// TIA Portal V17 export
// export: Created 2022-07-20T07:01:33.194346Z, ExportSetting WithDefaults, DisplayName Totally Integrated Automation Portal, DisplayVersion V17, DisplayName TIA Portal Openness, DisplayVersion V17, DisplayName TIA Portal Version Control Interface, DisplayVersion V17, DisplayName SINAMICS Startdrive Advanced, DisplayVersion V17, DisplayName SINAMICS Startdrive G130, G150, S120, S150, SINAMICS MV, S210, DisplayVersion V17, DisplayName SINAMICS Startdrive G110M, G120, G120C, G120D, G120P, G115D, DisplayVersion V17, DisplayName STEP 7 Professional, DisplayVersion V17, DisplayName STEP 7 Safety, DisplayVersion V17, DisplayName WinCC Advanced, DisplayVersion V17
FUNCTION_BLOCK "FB10321_CompactPrintingHeadsTray"   // FB10321, LAD
{ S7_Optimized_Access := 'TRUE' }
VERSION : 0.1
// stored: AutoNumber false, IsIECCheckEnabled false, IsRetainMemResEnabled false, MemoryReserve 100, SetENOAutomatically false, UDAEnableTagReadback false
   VAR_INPUT
      HeadsTray_RequestHeadsTraySafetyPosition : Bool;
      VerticalMotor_OriginPosition : Real;
      VerticalMotor_CleaningPosition : Real;
      VerticalMotor_WipingPosition : Real;
      VerticalMotor_PurgePosition : Real;
      VerticalMotor_PrintingPosition : Real;
      "VerticalMotor_Velocity_mm.s-1" : Real;
      VerticalMotor_ScaleInverted : Bool;
      HorizontalMotor_OriginPosition : Real;
      HorizontalMotor_WipingPosition : Real;
      HorizontalMotor_PurgePosition : Real;
      HorizontalMotor_Heads12Position : Real;
      HorizontalMotor_Heads34Position : Real;
      HorizontalMotor_Heads56Position : Real;
      HorizontalMotor_PrintingPosition : Real;
      "HorizontalMotor_Velocity_mm.s-1" : Real;
      HorizontalMotor_ScaleInverted : Bool;
      VerticalMotorDrive_In : "TLexium_MDrv_Drv2Plc";
      HorizontalMotorDrive_In : "TLexium_MDrv_Drv2Plc";
   END_VAR
   VAR_OUTPUT
      VerticalMotor_ActualPosition_mm : Real;
      HorizontalMotor_ActualPosition_mm : Real;
      HeadsTray_HomingDone : Bool;
      HeadsTray_IsInSafetyPosition : Bool;
      HeadsTray_IsInOriginPosition : Bool;
      HeadsTray_IsInHeads12CleaningPosition : Bool;
      HeadsTray_IsInHeads34CleaningPosition : Bool;
      HeadsTray_IsInHeads56CleaningPosition : Bool;
      HeadsTray_IsInWipingPosition : Bool;
      HeadsTray_IsInPurgePosition : Bool;
      HeadsTray_IsInHighPosition : Bool;
      HeadsTray_IsInPrintingPosition : Bool;
      HorizontalMotor_IsInOriginPosition : Bool;
      HorizontalMotor_IsInPurgePosition : Bool;
      HorizontalMotor_IsInWipingPosition : Bool;
      HorizontalMotor_IsInHeads12Position : Bool;
      HorizontalMotor_IsInHeads34Position : Bool;
      HorizontalMotor_IsInHeads56Position : Bool;
      HorizontalMotor_IsInPrintingPosition : Bool;
      VerticalMotor_IsInOriginPosition : Bool;
      VerticalMotor_IsInCleaningPosition : Bool;
      VerticalMotor_IsInWipingPosition : Bool;
      VerticalMotor_IsInPurgePosition : Bool;
      VerticalMotor_IsInPrintingPosition : Bool;
      SuccionDisk : Bool;
      VerticalMotor_InError : Bool;
      VerticalMotor_ErrorCode : Array[0..9] of UInt;
      HorizontalMotor_InError : Bool;
      HorizontalMotor_ErrorCode : Array[0..9] of UInt;
   END_VAR
   VAR_IN_OUT
      VerticalMotorDrive_Out : "TLexium_MDrv_Plc2Drv";
      HorizontalMotorDrive_Out : "TLexium_MDrv_Plc2Drv";
      RequestAcknowledge : Bool;
      RequestHoming : Bool;
      RequestStop : Bool;
      RequestGoToOriginPosition : Bool;
      RequestGoToWipingPosition : Bool;
      RequestGoToPurgePosition : Bool;
      RequestGoToHorizontalHeads12Position : Bool;
      RequestGoToHorizontalHeads34Position : Bool;
      RequestGoToHorizontalHeads56Position : Bool;
      RequestGoToVerticalOriginPosition : Bool;
      RequestGoToVerticalCleaningPosition : Bool;
      RequestGoToHighPosition : Bool;
      RequestGoToPrintingPosition : Bool;
   END_VAR
   VAR
      HeadsTrayMovementStateDiagram : Int;
      HeadsTraySafetyMovementStateDiagram : Int;
      R_TRIG_RequestHoming : R_TRIG;
      R_TRIG_RequestGoToOriginPosition { S7_SetPoint := 'True'} : R_TRIG;
      R_TRIG_RequestGoToWipingPosition { S7_SetPoint := 'True'} : R_TRIG;
      R_TRIG_RequestGoToPurgePosition { S7_SetPoint := 'True'} : R_TRIG;
      R_TRIG_RequestGoToHorizontalHeads12Position { S7_SetPoint := 'True'} : R_TRIG;
      R_TRIG_RequestGoToHorizontalHeads34Position { S7_SetPoint := 'True'} : R_TRIG;
      R_TRIG_RequestGoToHorizontalHeads56Position { S7_SetPoint := 'True'} : R_TRIG;
      R_TRIG_RequestGoToVerticalOriginPosition { S7_SetPoint := 'True'} : R_TRIG;
      R_TRIG_RequestGoToVerticalCleaningPosition { S7_SetPoint := 'True'} : R_TRIG;
      R_TRIG_RequestGoToHighPosition { S7_SetPoint := 'True'} : R_TRIG;
      R_TRIG_RequestGoToPrintingPosition { S7_SetPoint := 'True'} : R_TRIG;
      R_TRIG_VerticalMotorHomingDone { S7_SetPoint := 'True'} : R_TRIG;
      R_TRIG_HorizontalMotorHomingDone { S7_SetPoint := 'True'} : R_TRIG;
      R_TRIG_HeadsTrayRequestHeadsTraySafety { S7_SetPoint := 'True'} : R_TRIG;
      TON_SafetyAcknowledgeTimer { S7_SetPoint := 'True'} : TON_TIME;
      VerticalMotorStruct : Struct
         In : Struct
            RequestAcknowledge : Bool;
            RequestHoming : Bool;
            RequestStop : Bool;
            RequestGoToOriginPosition : Bool;
            RequestGoToCleaningPosition : Bool;
            RequestGoToWipingPosition : Bool;
            RequestGoToPurgePosition : Bool;
            RequestGoToPrintingPosition : Bool;
            OriginPosition : Real;
            CleaningPosition : Real;
            WipingPositon : Real;
            PurgePosition : Real;
            PrintingPosition : Real;
            "Velocity_mm.s-1" : Real;
            ScaleInverted : Bool;
         END_STRUCT;
         Out : Struct
            MotorInMovement : Bool;
            ActualPosition : Real;
            HomingDone : Bool;
            IsInOriginPosition : Bool;
            IsInCleaningPosition : Bool;
            IsInWipingPosition : Bool;
            IsInPurgePosition : Bool;
            IsInPrintingPosition : Bool;
            InError : Bool;
            ErrorCode : Array[0..9] of UInt;
         END_STRUCT;
      END_STRUCT;
      HorizontalMotorStruct : Struct
         In : Struct
            RequestAcknowledge : Bool;
            RequestHoming : Bool;
            RequestStop : Bool;
            RequestGoToOriginPosition : Bool;
            RequestGoToWipingPosition : Bool;
            RequestGoToPurgePosition : Bool;
            RequestGoToHeads12Position : Bool;
            RequestGoToHeads34Position : Bool;
            RequestGoToHeads56Position : Bool;
            RequestGoToPrintingPosition : Bool;
            OriginPosition : Real;
            WipingPositin : Real;
            PurgePosition : Real;
            Heads12Position : Real;
            Heads34Position : Real;
            Heads56Position : Real;
            PrintingPosition : Real;
            "Velocity_mm.s-1" : Real;
            ScaleInverted : Bool;
         END_STRUCT;
         Out : Struct
            MotorInMovement : Bool;
            ActualPosition : Real;
            HomingDone : Bool;
            IsInOriginPosition : Bool;
            IsInWipingPosition : Bool;
            IsInPurgePosition : Bool;
            IsInHeads12Position : Bool;
            IsInHeads34Position : Bool;
            IsInHeads56Position : Bool;
            IsInPrintingPosition : Bool;
            InError : Bool;
            ErrorCode : Array[0..9] of UInt;
         END_STRUCT;
      END_STRUCT;
      FB10234_LexiumMotor_Vertical { S7_SetPoint := 'True'} : "FB10234_LexiumMotor";
      FB10234_LexiumMotor_Horizontal { S7_SetPoint := 'True'} : "FB10234_LexiumMotor";
   END_VAR
   VAR CONSTANT
      "0_WAIT_FOR_MOTOR_HEADSTRAY_REQUESTS" : Int := 0;
      "10_HOMING_VERTICAL_MOTOR" : Int := 10;
      "11_HOMING_HORIZONTAL_MOTOR" : Int := 11;
      "20_ORIGIN_POSITION_VERTICAL" : Int := 20;
      "21_ORIGIN_POSITION_HORIZONTAL" : Int := 21;
      "30_WIPING_POSITION_VERTICAL_ORIGIN" : Int := 30;
      "31_WIPING_POSITION_HORIZONTAL" : Int := 31;
      "32_WIPING_POSITION_VERTICAL_WIPING" : Int := 32;
      "40_PURGE_POSITION_VERTICAL_ORIGIN" : Int := 40;
      "41_PURGE_POSITION_HORIZONTAL" : Int := 41;
      "42_PURGE_POSITION_VERTICAL_PURGE" : Int := 42;
      "50_HEADS12_POSITION_VERTICAL_ORIGIN" : Int := 50;
      "51_HEADS12_POSITION_HORIZONTAL" : Int := 51;
      "60_HEADS34_POSITION_VERTICAL_ORIGIN" : Int := 60;
      "61_HEADS34_POSITION_HORIZONTAL" : Int := 61;
      "70_HEADS56_POSITION_VERTICAL_ORIGIN" : Int := 70;
      "71_HEADS56_POSITION_HORIZONTAL" : Int := 71;
      "80_HIGH_POSITION_VERTICAL_ORIGIN" : Int := 80;
      "81_HIGH_POSITION_HORIZONTAL_PRINTING" : Int := 81;
      "90_PRINT_POSITION_VERTICAL_ORIGIN" : Int := 90;
      "91_PRINT_POSITION_HORIZONTAL_PRINTING" : Int := 91;
      "92_PRINT_POSITION_VERTICAL_PRINTING" : Int := 92;
      "100_VERTICAL_ORIGIN" : Int := 100;
      "110_VERTICAL_CLEANING" : Int := 110;
      "10000_MOTOR_HEADSTRAY_REQUEST_DONE" : Int := 10000;
      "==========" : Bool;
      "0_WAIT_FOR_SAFETY_MOVEMENT" : Int := 0;
      "10_SAFETY_STOP" : Int := 10;
      "20_SAFETY_ACKNWOLEDGE" : Int := 20;
      "30_SAFETY_HOMING_VERTICAL_MOTOR" : Int := 30;
      "31_SAFETY_HOMING_HORIZONTAL_MOTOR" : Int := 31;
      "40_SAFETY_VERTICAL_MOTOR_ORIGIN" : Int := 40;
      "41_SAFETY_HORIZONTAL_MOTOR_ORIGIN" : Int := 41;
      "10000_SAFETY_MOVEMENT_DONE" : Int := 10000;
   END_VAR
BEGIN

REGION Network 1 (SCL): FirstScan
   IF "FirstScan" THEN
       #HeadsTray_HomingDone := FALSE;
       #HeadsTray_IsInOriginPosition := FALSE;
       #HeadsTray_IsInWipingPosition := FALSE;
       #HeadsTray_IsInHeads12CleaningPosition := FALSE;
       #HeadsTray_IsInHeads34CleaningPosition := FALSE;
       #HeadsTray_IsInHeads56CleaningPosition := FALSE;
       #HeadsTray_IsInPurgePosition := FALSE;
       #HeadsTray_IsInHighPosition := FALSE;
       #HeadsTray_IsInPrintingPosition := FALSE;

       #HorizontalMotorStruct.In.RequestGoToOriginPosition := FALSE;
       #HorizontalMotorStruct.In.RequestGoToWipingPosition := FALSE;
       #HorizontalMotorStruct.In.RequestGoToPurgePosition := FALSE;
       #HorizontalMotorStruct.In.RequestGoToHeads12Position := FALSE;
       #HorizontalMotorStruct.In.RequestGoToHeads34Position := FALSE;
       #HorizontalMotorStruct.In.RequestGoToHeads56Position := FALSE;
       #HorizontalMotorStruct.In.RequestGoToPrintingPosition := FALSE;
       #HorizontalMotor_IsInOriginPosition := FALSE;
       #HorizontalMotor_IsInPurgePosition := FALSE;
       #HorizontalMotor_IsInHeads12Position := FALSE;
       #HorizontalMotor_IsInHeads34Position := FALSE;
       #HorizontalMotor_IsInHeads56Position := FALSE;
       #HorizontalMotor_IsInPrintingPosition := FALSE;

       #VerticalMotorStruct.In.RequestGoToOriginPosition := FALSE;
       #VerticalMotorStruct.In.RequestGoToCleaningPosition := FALSE;
       #VerticalMotorStruct.In.RequestGoToWipingPosition := FALSE;
       #VerticalMotorStruct.In.RequestGoToPurgePosition := FALSE;
       #VerticalMotorStruct.In.RequestGoToPrintingPosition := FALSE;
       #VerticalMotor_IsInOriginPosition := FALSE;
       #VerticalMotor_IsInCleaningPosition := FALSE;
       #VerticalMotor_IsInWipingPosition := FALSE;
       #VerticalMotor_IsInPurgePosition := FALSE;
       #VerticalMotor_IsInPrintingPosition := FALSE;

       #HeadsTrayMovementStateDiagram := #"0_WAIT_FOR_MOTOR_HEADSTRAY_REQUESTS";
   END_IF;
END_REGION

REGION Network 2 (SCL): Edge Signal & Timers
   REGION EDGE SIGNAL
       #R_TRIG_RequestHoming(CLK := #RequestHoming AND #HeadsTrayMovementStateDiagram = #"0_WAIT_FOR_MOTOR_HEADSTRAY_REQUESTS");
       #R_TRIG_VerticalMotorHomingDone(CLK := #VerticalMotorStruct.Out.HomingDone);
       #R_TRIG_HorizontalMotorHomingDone(CLK := #HorizontalMotorStruct.Out.HomingDone);

       #R_TRIG_RequestGoToOriginPosition(CLK := #RequestGoToOriginPosition AND #HeadsTrayMovementStateDiagram = #"0_WAIT_FOR_MOTOR_HEADSTRAY_REQUESTS" AND NOT (#HeadsTray_IsInOriginPosition));
       #R_TRIG_RequestGoToWipingPosition(CLK := #RequestGoToWipingPosition AND #HeadsTrayMovementStateDiagram = #"0_WAIT_FOR_MOTOR_HEADSTRAY_REQUESTS" AND NOT (#HeadsTray_IsInWipingPosition));
       #R_TRIG_RequestGoToPurgePosition(CLK := #RequestGoToPurgePosition AND #HeadsTrayMovementStateDiagram = #"0_WAIT_FOR_MOTOR_HEADSTRAY_REQUESTS" AND NOT (#HeadsTray_IsInPurgePosition));
       #R_TRIG_RequestGoToHorizontalHeads12Position(CLK := #RequestGoToHorizontalHeads12Position AND #HeadsTrayMovementStateDiagram = #"0_WAIT_FOR_MOTOR_HEADSTRAY_REQUESTS" AND NOT (#HorizontalMotor_IsInHeads12Position));
       #R_TRIG_RequestGoToHorizontalHeads34Position(CLK := #RequestGoToHorizontalHeads34Position AND #HeadsTrayMovementStateDiagram = #"0_WAIT_FOR_MOTOR_HEADSTRAY_REQUESTS" AND NOT (#HorizontalMotor_IsInHeads34Position));
       #R_TRIG_RequestGoToHorizontalHeads56Position(CLK := #RequestGoToHorizontalHeads56Position AND #HeadsTrayMovementStateDiagram = #"0_WAIT_FOR_MOTOR_HEADSTRAY_REQUESTS" AND NOT (#HorizontalMotor_IsInHeads56Position));
       #R_TRIG_RequestGoToVerticalCleaningPosition(CLK := #RequestGoToVerticalCleaningPosition AND #HeadsTrayMovementStateDiagram = #"0_WAIT_FOR_MOTOR_HEADSTRAY_REQUESTS" AND NOT (#HeadsTray_IsInHeads12CleaningPosition AND #HeadsTray_IsInHeads34CleaningPosition AND #HeadsTray_IsInHeads56CleaningPosition));
       #R_TRIG_RequestGoToHighPosition(CLK := #RequestGoToHighPosition AND #HeadsTrayMovementStateDiagram = #"0_WAIT_FOR_MOTOR_HEADSTRAY_REQUESTS" AND NOT (#HeadsTray_IsInHighPosition));
       #R_TRIG_RequestGoToPrintingPosition(CLK := #RequestGoToPrintingPosition AND #HeadsTrayMovementStateDiagram = #"0_WAIT_FOR_MOTOR_HEADSTRAY_REQUESTS" AND NOT (#HeadsTray_IsInPrintingPosition));
       #R_TRIG_HeadsTrayRequestHeadsTraySafety(CLK := #HeadsTray_RequestHeadsTraySafetyPosition);
       #R_TRIG_RequestGoToVerticalOriginPosition(CLK := #RequestGoToVerticalOriginPosition AND #HeadsTrayMovementStateDiagram = #"0_WAIT_FOR_MOTOR_HEADSTRAY_REQUESTS" AND NOT (#VerticalMotor_IsInOriginPosition));
   END_REGION

   REGION TIMERS
       #TON_SafetyAcknowledgeTimer(IN := #HeadsTraySafetyMovementStateDiagram = #"20_SAFETY_ACKNWOLEDGE",
                                   PT := T#2s);
   END_REGION
END_REGION

REGION Network 3 (SCL): HeadsTray Commands Management
   REGION MOTORS PARAMETERS
       #VerticalMotorStruct.In.RequestAcknowledge := #HorizontalMotorStruct.In.RequestAcknowledge := #RequestAcknowledge;
       #VerticalMotorStruct.In.RequestStop := #RequestStop;
       #HorizontalMotorStruct.In.RequestStop := #RequestStop;

       #VerticalMotorStruct.In."Velocity_mm.s-1" := #"VerticalMotor_Velocity_mm.s-1";
       #VerticalMotorStruct.In.ScaleInverted := #VerticalMotor_ScaleInverted;

       #HorizontalMotorStruct.In."Velocity_mm.s-1" := #"HorizontalMotor_Velocity_mm.s-1";
       #HorizontalMotorStruct.In.ScaleInverted := #HorizontalMotor_ScaleInverted;
   END_REGION

   REGION VERTICAL MOTOR POSITION PARAMETERS
       #VerticalMotorStruct.In.OriginPosition := #VerticalMotor_OriginPosition;
       #VerticalMotorStruct.In.PurgePosition := #VerticalMotor_PurgePosition;
       #VerticalMotorStruct.In.CleaningPosition := #VerticalMotor_CleaningPosition;
       #VerticalMotorStruct.In.WipingPositon := #VerticalMotor_WipingPosition;
       #VerticalMotorStruct.In.PrintingPosition := #VerticalMotor_PrintingPosition;
   END_REGION

   REGION HORIZONTAL MOTOR POSITION PARAMETERS
       #HorizontalMotorStruct.In.OriginPosition := #HorizontalMotor_OriginPosition;
       #HorizontalMotorStruct.In.WipingPositin := #HorizontalMotor_WipingPosition;
       #HorizontalMotorStruct.In.PurgePosition := #HorizontalMotor_PurgePosition;
       #HorizontalMotorStruct.In.Heads12Position := #HorizontalMotor_Heads12Position;
       #HorizontalMotorStruct.In.Heads34Position := #HorizontalMotor_Heads34Position;
       #HorizontalMotorStruct.In.Heads56Position := #HorizontalMotor_Heads56Position;
       #HorizontalMotorStruct.In.PrintingPosition := #HorizontalMotor_PrintingPosition;
   END_REGION
END_REGION

REGION Network 4: Vertical Motor Management
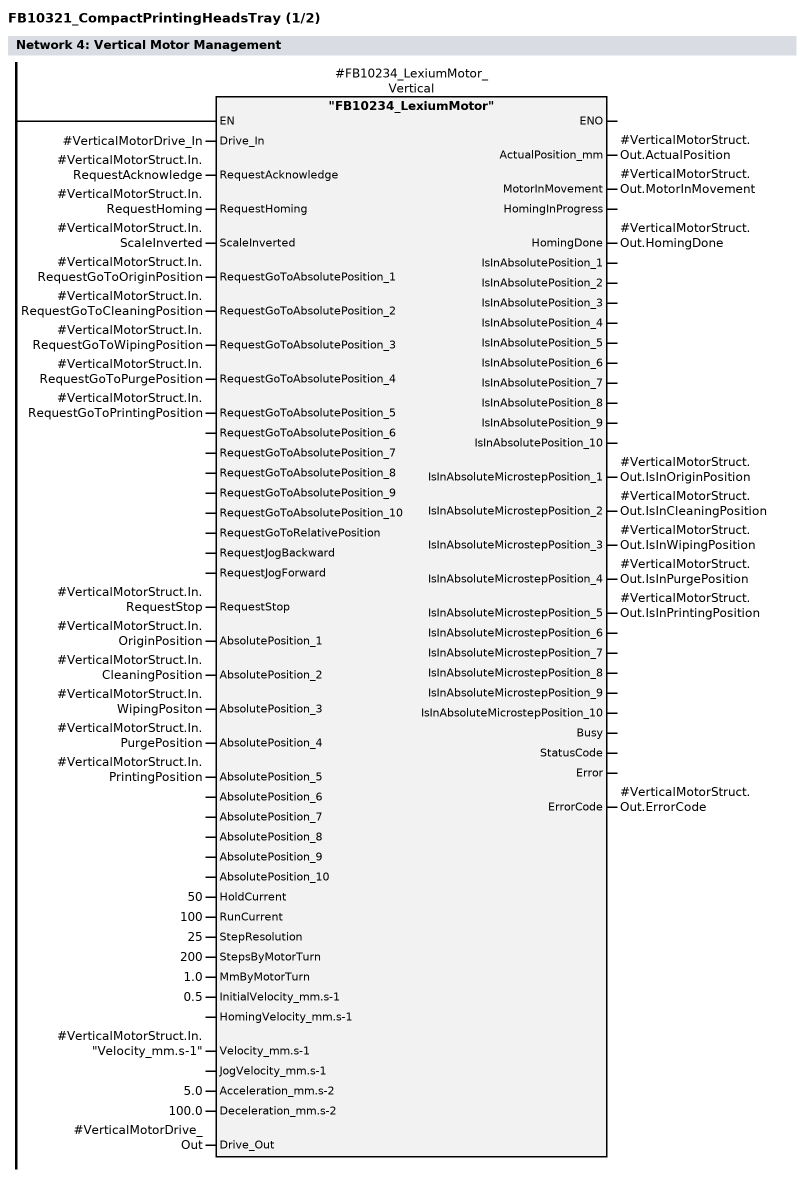
   RUNG wire#powerrail
      #FB10234_LexiumMotor_Vertical(Drive_In := #VerticalMotorDrive_In, RequestAcknowledge := #VerticalMotorStruct.In.RequestAcknowledge, RequestHoming := #VerticalMotorStruct.In.RequestHoming, ScaleInverted := #VerticalMotorStruct.In.ScaleInverted, RequestGoToAbsolutePosition_1 := #VerticalMotorStruct.In.RequestGoToOriginPosition, RequestGoToAbsolutePosition_2 := #VerticalMotorStruct.In.RequestGoToCleaningPosition, RequestGoToAbsolutePosition_3 := #VerticalMotorStruct.In.RequestGoToWipingPosition, RequestGoToAbsolutePosition_4 := #VerticalMotorStruct.In.RequestGoToPurgePosition, RequestGoToAbsolutePosition_5 := #VerticalMotorStruct.In.RequestGoToPrintingPosition, RequestGoToAbsolutePosition_6 :=, RequestGoToAbsolutePosition_7 :=, RequestGoToAbsolutePosition_8 :=, RequestGoToAbsolutePosition_9 :=, RequestGoToAbsolutePosition_10 :=, RequestGoToRelativePosition :=, RequestJogBackward :=, RequestJogForward :=, RequestStop := #VerticalMotorStruct.In.RequestStop, AbsolutePosition_1 := #VerticalMotorStruct.In.OriginPosition, AbsolutePosition_2 := #VerticalMotorStruct.In.CleaningPosition, AbsolutePosition_3 := #VerticalMotorStruct.In.WipingPositon, AbsolutePosition_4 := #VerticalMotorStruct.In.PurgePosition, AbsolutePosition_5 := #VerticalMotorStruct.In.PrintingPosition, AbsolutePosition_6 :=, AbsolutePosition_7 :=, AbsolutePosition_8 :=, AbsolutePosition_9 :=, AbsolutePosition_10 :=, HoldCurrent := 50, RunCurrent := 100, StepResolution := 25, StepsByMotorTurn := 200, MmByMotorTurn := 1.0, "InitialVelocity_mm.s-1" := 0.5, "HomingVelocity_mm.s-1" :=, "Velocity_mm.s-1" := #VerticalMotorStruct.In."Velocity_mm.s-1", "JogVelocity_mm.s-1" :=, "Acceleration_mm.s-2" := 5.0, "Deceleration_mm.s-2" := 100.0, Drive_Out := #VerticalMotorDrive_Out, ActualPosition_mm => #VerticalMotorStruct.Out.ActualPosition, MotorInMovement => #VerticalMotorStruct.Out.MotorInMovement, HomingInProgress =>, HomingDone => #VerticalMotorStruct.Out.HomingDone, IsInAbsolutePosition_1 =>, IsInAbsolutePosition_2 =>, IsInAbsolutePosition_3 =>, IsInAbsolutePosition_4 =>, IsInAbsolutePosition_5 =>, IsInAbsolutePosition_6 =>, IsInAbsolutePosition_7 =>, IsInAbsolutePosition_8 =>, IsInAbsolutePosition_9 =>, IsInAbsolutePosition_10 =>, IsInAbsoluteMicrostepPosition_1 => #VerticalMotorStruct.Out.IsInOriginPosition, IsInAbsoluteMicrostepPosition_2 => #VerticalMotorStruct.Out.IsInCleaningPosition, IsInAbsoluteMicrostepPosition_3 => #VerticalMotorStruct.Out.IsInWipingPosition, IsInAbsoluteMicrostepPosition_4 => #VerticalMotorStruct.Out.IsInPurgePosition, IsInAbsoluteMicrostepPosition_5 => #VerticalMotorStruct.Out.IsInPrintingPosition, IsInAbsoluteMicrostepPosition_6 =>, IsInAbsoluteMicrostepPosition_7 =>, IsInAbsoluteMicrostepPosition_8 =>, IsInAbsoluteMicrostepPosition_9 =>, IsInAbsoluteMicrostepPosition_10 =>, Busy =>, StatusCode =>, Error =>, ErrorCode => #VerticalMotorStruct.Out.ErrorCode)
   END_RUNG
   // the same network as SCL:
   #FB10234_LexiumMotor_Vertical(Drive_In := #VerticalMotorDrive_In,   // "FB10234_LexiumMotor"
                           RequestAcknowledge := #VerticalMotorStruct.In.RequestAcknowledge,
                           RequestHoming := #VerticalMotorStruct.In.RequestHoming,
                           ScaleInverted := #VerticalMotorStruct.In.ScaleInverted,
                           RequestGoToAbsolutePosition_1 := #VerticalMotorStruct.In.RequestGoToOriginPosition,
                           RequestGoToAbsolutePosition_2 := #VerticalMotorStruct.In.RequestGoToCleaningPosition,
                           RequestGoToAbsolutePosition_3 := #VerticalMotorStruct.In.RequestGoToWipingPosition,
                           RequestGoToAbsolutePosition_4 := #VerticalMotorStruct.In.RequestGoToPurgePosition,
                           RequestGoToAbsolutePosition_5 := #VerticalMotorStruct.In.RequestGoToPrintingPosition,
                           RequestStop := #VerticalMotorStruct.In.RequestStop,
                           AbsolutePosition_1 := #VerticalMotorStruct.In.OriginPosition,
                           AbsolutePosition_2 := #VerticalMotorStruct.In.CleaningPosition,
                           AbsolutePosition_3 := #VerticalMotorStruct.In.WipingPositon,
                           AbsolutePosition_4 := #VerticalMotorStruct.In.PurgePosition,
                           AbsolutePosition_5 := #VerticalMotorStruct.In.PrintingPosition,
                           HoldCurrent := 50,
                           RunCurrent := 100,
                           StepResolution := 25,
                           StepsByMotorTurn := 200,
                           MmByMotorTurn := 1.0,
                           "InitialVelocity_mm.s-1" := 0.5,
                           "Velocity_mm.s-1" := #VerticalMotorStruct.In."Velocity_mm.s-1",
                           "Acceleration_mm.s-2" := 5.0,
                           "Deceleration_mm.s-2" := 100.0,
                           Drive_Out := #VerticalMotorDrive_Out,
                           ActualPosition_mm => #VerticalMotorStruct.Out.ActualPosition,
                           MotorInMovement => #VerticalMotorStruct.Out.MotorInMovement,
                           HomingDone => #VerticalMotorStruct.Out.HomingDone,
                           IsInAbsoluteMicrostepPosition_1 => #VerticalMotorStruct.Out.IsInOriginPosition,
                           IsInAbsoluteMicrostepPosition_2 => #VerticalMotorStruct.Out.IsInCleaningPosition,
                           IsInAbsoluteMicrostepPosition_3 => #VerticalMotorStruct.Out.IsInWipingPosition,
                           IsInAbsoluteMicrostepPosition_4 => #VerticalMotorStruct.Out.IsInPurgePosition,
                           IsInAbsoluteMicrostepPosition_5 => #VerticalMotorStruct.Out.IsInPrintingPosition,
                           ErrorCode => #VerticalMotorStruct.Out.ErrorCode);
END_REGION

REGION Network 5: Horizontal Motor Management
   // 50.24
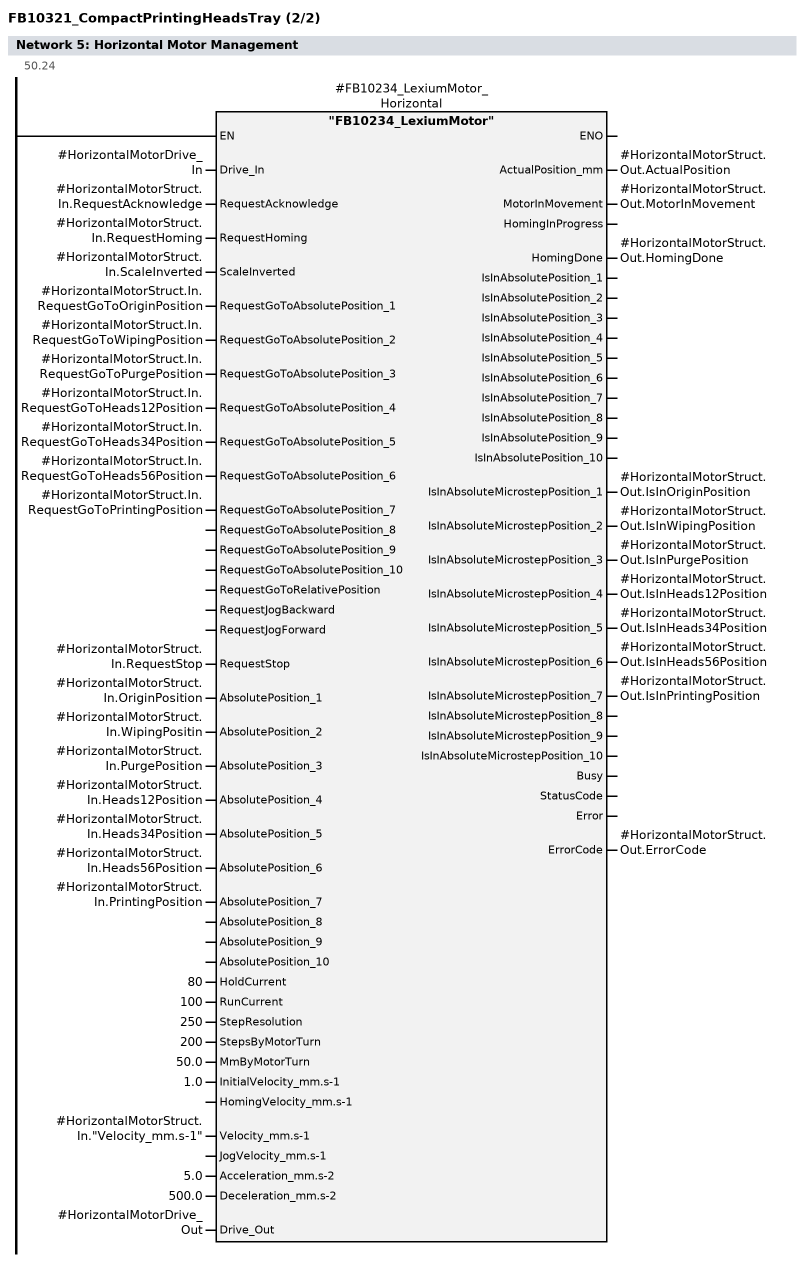
   RUNG wire#powerrail
      #FB10234_LexiumMotor_Horizontal(Drive_In := #HorizontalMotorDrive_In, RequestAcknowledge := #HorizontalMotorStruct.In.RequestAcknowledge, RequestHoming := #HorizontalMotorStruct.In.RequestHoming, ScaleInverted := #HorizontalMotorStruct.In.ScaleInverted, RequestGoToAbsolutePosition_1 := #HorizontalMotorStruct.In.RequestGoToOriginPosition, RequestGoToAbsolutePosition_2 := #HorizontalMotorStruct.In.RequestGoToWipingPosition, RequestGoToAbsolutePosition_3 := #HorizontalMotorStruct.In.RequestGoToPurgePosition, RequestGoToAbsolutePosition_4 := #HorizontalMotorStruct.In.RequestGoToHeads12Position, RequestGoToAbsolutePosition_5 := #HorizontalMotorStruct.In.RequestGoToHeads34Position, RequestGoToAbsolutePosition_6 := #HorizontalMotorStruct.In.RequestGoToHeads56Position, RequestGoToAbsolutePosition_7 := #HorizontalMotorStruct.In.RequestGoToPrintingPosition, RequestGoToAbsolutePosition_8 :=, RequestGoToAbsolutePosition_9 :=, RequestGoToAbsolutePosition_10 :=, RequestGoToRelativePosition :=, RequestJogBackward :=, RequestJogForward :=, RequestStop := #HorizontalMotorStruct.In.RequestStop, AbsolutePosition_1 := #HorizontalMotorStruct.In.OriginPosition, AbsolutePosition_2 := #HorizontalMotorStruct.In.WipingPositin, AbsolutePosition_3 := #HorizontalMotorStruct.In.PurgePosition, AbsolutePosition_4 := #HorizontalMotorStruct.In.Heads12Position, AbsolutePosition_5 := #HorizontalMotorStruct.In.Heads34Position, AbsolutePosition_6 := #HorizontalMotorStruct.In.Heads56Position, AbsolutePosition_7 := #HorizontalMotorStruct.In.PrintingPosition, AbsolutePosition_8 :=, AbsolutePosition_9 :=, AbsolutePosition_10 :=, HoldCurrent := 80, RunCurrent := 100, StepResolution := 250, StepsByMotorTurn := 200, MmByMotorTurn := 50.0, "InitialVelocity_mm.s-1" := 1.0, "HomingVelocity_mm.s-1" :=, "Velocity_mm.s-1" := #HorizontalMotorStruct.In."Velocity_mm.s-1", "JogVelocity_mm.s-1" :=, "Acceleration_mm.s-2" := 5.0, "Deceleration_mm.s-2" := 500.0, Drive_Out := #HorizontalMotorDrive_Out, ActualPosition_mm => #HorizontalMotorStruct.Out.ActualPosition, MotorInMovement => #HorizontalMotorStruct.Out.MotorInMovement, HomingInProgress =>, HomingDone => #HorizontalMotorStruct.Out.HomingDone, IsInAbsolutePosition_1 =>, IsInAbsolutePosition_2 =>, IsInAbsolutePosition_3 =>, IsInAbsolutePosition_4 =>, IsInAbsolutePosition_5 =>, IsInAbsolutePosition_6 =>, IsInAbsolutePosition_7 =>, IsInAbsolutePosition_8 =>, IsInAbsolutePosition_9 =>, IsInAbsolutePosition_10 =>, IsInAbsoluteMicrostepPosition_1 => #HorizontalMotorStruct.Out.IsInOriginPosition, IsInAbsoluteMicrostepPosition_2 => #HorizontalMotorStruct.Out.IsInWipingPosition, IsInAbsoluteMicrostepPosition_3 => #HorizontalMotorStruct.Out.IsInPurgePosition, IsInAbsoluteMicrostepPosition_4 => #HorizontalMotorStruct.Out.IsInHeads12Position, IsInAbsoluteMicrostepPosition_5 => #HorizontalMotorStruct.Out.IsInHeads34Position, IsInAbsoluteMicrostepPosition_6 => #HorizontalMotorStruct.Out.IsInHeads56Position, IsInAbsoluteMicrostepPosition_7 => #HorizontalMotorStruct.Out.IsInPrintingPosition, IsInAbsoluteMicrostepPosition_8 =>, IsInAbsoluteMicrostepPosition_9 =>, IsInAbsoluteMicrostepPosition_10 =>, Busy =>, StatusCode =>, Error =>, ErrorCode => #HorizontalMotorStruct.Out.ErrorCode)
   END_RUNG
   // the same network as SCL:
   #FB10234_LexiumMotor_Horizontal(Drive_In := #HorizontalMotorDrive_In,   // "FB10234_LexiumMotor"
                           RequestAcknowledge := #HorizontalMotorStruct.In.RequestAcknowledge,
                           RequestHoming := #HorizontalMotorStruct.In.RequestHoming,
                           ScaleInverted := #HorizontalMotorStruct.In.ScaleInverted,
                           RequestGoToAbsolutePosition_1 := #HorizontalMotorStruct.In.RequestGoToOriginPosition,
                           RequestGoToAbsolutePosition_2 := #HorizontalMotorStruct.In.RequestGoToWipingPosition,
                           RequestGoToAbsolutePosition_3 := #HorizontalMotorStruct.In.RequestGoToPurgePosition,
                           RequestGoToAbsolutePosition_4 := #HorizontalMotorStruct.In.RequestGoToHeads12Position,
                           RequestGoToAbsolutePosition_5 := #HorizontalMotorStruct.In.RequestGoToHeads34Position,
                           RequestGoToAbsolutePosition_6 := #HorizontalMotorStruct.In.RequestGoToHeads56Position,
                           RequestGoToAbsolutePosition_7 := #HorizontalMotorStruct.In.RequestGoToPrintingPosition,
                           RequestStop := #HorizontalMotorStruct.In.RequestStop,
                           AbsolutePosition_1 := #HorizontalMotorStruct.In.OriginPosition,
                           AbsolutePosition_2 := #HorizontalMotorStruct.In.WipingPositin,
                           AbsolutePosition_3 := #HorizontalMotorStruct.In.PurgePosition,
                           AbsolutePosition_4 := #HorizontalMotorStruct.In.Heads12Position,
                           AbsolutePosition_5 := #HorizontalMotorStruct.In.Heads34Position,
                           AbsolutePosition_6 := #HorizontalMotorStruct.In.Heads56Position,
                           AbsolutePosition_7 := #HorizontalMotorStruct.In.PrintingPosition,
                           HoldCurrent := 80,
                           RunCurrent := 100,
                           StepResolution := 250,
                           StepsByMotorTurn := 200,
                           MmByMotorTurn := 50.0,
                           "InitialVelocity_mm.s-1" := 1.0,
                           "Velocity_mm.s-1" := #HorizontalMotorStruct.In."Velocity_mm.s-1",
                           "Acceleration_mm.s-2" := 5.0,
                           "Deceleration_mm.s-2" := 500.0,
                           Drive_Out := #HorizontalMotorDrive_Out,
                           ActualPosition_mm => #HorizontalMotorStruct.Out.ActualPosition,
                           MotorInMovement => #HorizontalMotorStruct.Out.MotorInMovement,
                           HomingDone => #HorizontalMotorStruct.Out.HomingDone,
                           IsInAbsoluteMicrostepPosition_1 => #HorizontalMotorStruct.Out.IsInOriginPosition,
                           IsInAbsoluteMicrostepPosition_2 => #HorizontalMotorStruct.Out.IsInWipingPosition,
                           IsInAbsoluteMicrostepPosition_3 => #HorizontalMotorStruct.Out.IsInPurgePosition,
                           IsInAbsoluteMicrostepPosition_4 => #HorizontalMotorStruct.Out.IsInHeads12Position,
                           IsInAbsoluteMicrostepPosition_5 => #HorizontalMotorStruct.Out.IsInHeads34Position,
                           IsInAbsoluteMicrostepPosition_6 => #HorizontalMotorStruct.Out.IsInHeads56Position,
                           IsInAbsoluteMicrostepPosition_7 => #HorizontalMotorStruct.Out.IsInPrintingPosition,
                           ErrorCode => #HorizontalMotorStruct.Out.ErrorCode);
END_REGION

REGION Network 6 (SCL): Printing Heads Tray Safety Management
   IF #HeadsTraySafetyMovementStateDiagram > 0 THEN
       #HeadsTrayMovementStateDiagram := #"0_WAIT_FOR_MOTOR_HEADSTRAY_REQUESTS";
   END_IF;

   CASE #HeadsTraySafetyMovementStateDiagram OF
       #"0_WAIT_FOR_SAFETY_MOVEMENT":
           IF #R_TRIG_HeadsTrayRequestHeadsTraySafety.Q THEN
               #HeadsTraySafetyMovementStateDiagram := #"10_SAFETY_STOP";
           END_IF;
       #"10_SAFETY_STOP":
           #RequestStop := TRUE;

           IF NOT(#HorizontalMotorStruct.Out.MotorInMovement OR #VerticalMotorStruct.Out.MotorInMovement) THEN
               #RequestStop := TRUE;
               #HeadsTraySafetyMovementStateDiagram := #"20_SAFETY_ACKNWOLEDGE";
           END_IF;
       #"20_SAFETY_ACKNWOLEDGE":
           #RequestAcknowledge := "Clock_0.5Hz";

           IF NOT (#HorizontalMotorStruct.Out.InError OR #VerticalMotorStruct.Out.InError) THEN
               #RequestAcknowledge := FALSE;
               IF NOT (#HeadsTray_HomingDone) THEN
                   #HeadsTraySafetyMovementStateDiagram := #"30_SAFETY_HOMING_VERTICAL_MOTOR";
               ELSE
                   #HeadsTraySafetyMovementStateDiagram := #"40_SAFETY_VERTICAL_MOTOR_ORIGIN";
               END_IF;
           END_IF;
       #"30_SAFETY_HOMING_VERTICAL_MOTOR":
           #VerticalMotorStruct.In.RequestHoming := TRUE;
           IF #R_TRIG_VerticalMotorHomingDone.Q THEN
               #VerticalMotorStruct.In.RequestHoming := FALSE;
               #HeadsTraySafetyMovementStateDiagram := #"31_SAFETY_HOMING_HORIZONTAL_MOTOR";
           END_IF;
       #"31_SAFETY_HOMING_HORIZONTAL_MOTOR":
           #HorizontalMotorStruct.In.RequestHoming := TRUE;
           IF #R_TRIG_HorizontalMotorHomingDone.Q THEN
               #HorizontalMotorStruct.In.RequestHoming := FALSE;
               #HeadsTraySafetyMovementStateDiagram := #"10000_SAFETY_MOVEMENT_DONE";
           END_IF;

       #"40_SAFETY_VERTICAL_MOTOR_ORIGIN":
           #VerticalMotorStruct.In.RequestGoToOriginPosition := TRUE;
           IF #VerticalMotorStruct.Out.IsInOriginPosition THEN
               #VerticalMotorStruct.In.RequestGoToOriginPosition := FALSE;
               #HeadsTraySafetyMovementStateDiagram := #"41_SAFETY_HORIZONTAL_MOTOR_ORIGIN";
           END_IF;
       #"41_SAFETY_HORIZONTAL_MOTOR_ORIGIN":
           #HorizontalMotorStruct.In.RequestGoToOriginPosition := TRUE;
           IF #HorizontalMotorStruct.Out.IsInOriginPosition THEN
               #HorizontalMotorStruct.In.RequestGoToOriginPosition := FALSE;
               #HeadsTraySafetyMovementStateDiagram := #"10000_SAFETY_MOVEMENT_DONE";
           END_IF;
       #"10000_SAFETY_MOVEMENT_DONE":
           IF NOT (#HeadsTray_RequestHeadsTraySafetyPosition) THEN
               #HeadsTraySafetyMovementStateDiagram := #"0_WAIT_FOR_SAFETY_MOVEMENT";
           END_IF;
   END_CASE;
END_REGION

REGION Network 7 (SCL): Printing HeadsTray Management
   IF #RequestStop OR #VerticalMotor_InError OR #HorizontalMotor_InError THEN
       #HeadsTrayMovementStateDiagram := #"10000_MOTOR_HEADSTRAY_REQUEST_DONE";
   END_IF;

   CASE #HeadsTrayMovementStateDiagram OF
       #"0_WAIT_FOR_MOTOR_HEADSTRAY_REQUESTS":
           IF #R_TRIG_RequestHoming.Q THEN
               #SuccionDisk := FALSE;
               #HeadsTrayMovementStateDiagram := #"10_HOMING_VERTICAL_MOTOR";
           ELSIF #HeadsTray_HomingDone THEN
               IF #R_TRIG_RequestGoToOriginPosition.Q THEN
                   #SuccionDisk := FALSE;
                   #HeadsTrayMovementStateDiagram := #"20_ORIGIN_POSITION_VERTICAL";
               ELSIF #R_TRIG_RequestGoToWipingPosition.Q THEN
                   #SuccionDisk := FALSE;
                   #HeadsTrayMovementStateDiagram := #"30_WIPING_POSITION_VERTICAL_ORIGIN";
               ELSIF  #R_TRIG_RequestGoToPurgePosition.Q THEN
                   #SuccionDisk := TRUE;
                   #HeadsTrayMovementStateDiagram := #"40_PURGE_POSITION_VERTICAL_ORIGIN";
               ELSIF #R_TRIG_RequestGoToHorizontalHeads12Position.Q THEN
                   #SuccionDisk := FALSE;
                   #HeadsTrayMovementStateDiagram := #"50_HEADS12_POSITION_VERTICAL_ORIGIN";
               ELSIF #R_TRIG_RequestGoToHorizontalHeads34Position.Q  THEN
                   #SuccionDisk := FALSE;
                   #HeadsTrayMovementStateDiagram := #"60_HEADS34_POSITION_VERTICAL_ORIGIN";
               ELSIF #R_TRIG_RequestGoToHorizontalHeads56Position.Q THEN
                   #SuccionDisk := FALSE;
                   #HeadsTrayMovementStateDiagram := #"70_HEADS56_POSITION_VERTICAL_ORIGIN";
               ELSIF #R_TRIG_RequestGoToHighPosition.Q THEN
                   #SuccionDisk := FALSE;
                   #HeadsTrayMovementStateDiagram := #"80_HIGH_POSITION_VERTICAL_ORIGIN";
               ELSIF #R_TRIG_RequestGoToPrintingPosition.Q THEN
                   #SuccionDisk := FALSE;
                   #HeadsTrayMovementStateDiagram := #"90_PRINT_POSITION_VERTICAL_ORIGIN";
               END_IF;
           END_IF;
       #"10_HOMING_VERTICAL_MOTOR":
           #VerticalMotorStruct.In.RequestHoming := TRUE;
           IF #R_TRIG_VerticalMotorHomingDone.Q THEN
               #VerticalMotorStruct.In.RequestHoming := FALSE;
               #HeadsTrayMovementStateDiagram := #"11_HOMING_HORIZONTAL_MOTOR";
           END_IF;
       #"11_HOMING_HORIZONTAL_MOTOR":
           #HorizontalMotorStruct.In.RequestHoming := TRUE;
           IF #R_TRIG_HorizontalMotorHomingDone.Q THEN
               #HorizontalMotorStruct.In.RequestHoming := FALSE;
               #HeadsTrayMovementStateDiagram := #"10000_MOTOR_HEADSTRAY_REQUEST_DONE";
           END_IF;

       #"20_ORIGIN_POSITION_VERTICAL":
           #VerticalMotorStruct.In.RequestGoToOriginPosition := TRUE;
           IF #VerticalMotorStruct.Out.IsInOriginPosition THEN
               #VerticalMotorStruct.In.RequestGoToOriginPosition := FALSE;
               #HeadsTrayMovementStateDiagram := #"21_ORIGIN_POSITION_HORIZONTAL";
           END_IF;
       #"21_ORIGIN_POSITION_HORIZONTAL":
           #HorizontalMotorStruct.In.RequestGoToOriginPosition := TRUE;
           IF #HorizontalMotorStruct.Out.IsInOriginPosition THEN
               #HorizontalMotorStruct.In.RequestGoToOriginPosition := FALSE;
               #HeadsTrayMovementStateDiagram := #"10000_MOTOR_HEADSTRAY_REQUEST_DONE";
           END_IF;

       #"30_WIPING_POSITION_VERTICAL_ORIGIN":
           #VerticalMotorStruct.In.RequestGoToOriginPosition := TRUE;
           IF #VerticalMotorStruct.Out.IsInOriginPosition THEN
               #VerticalMotorStruct.In.RequestGoToOriginPosition := FALSE;
               #HeadsTrayMovementStateDiagram := #"21_ORIGIN_POSITION_HORIZONTAL";
           END_IF;
       #"31_WIPING_POSITION_HORIZONTAL":
           #HorizontalMotorStruct.In.RequestGoToWipingPosition := TRUE;
           IF #HorizontalMotorStruct.Out.IsInWipingPosition THEN
               #HorizontalMotorStruct.In.RequestGoToWipingPosition := FALSE;
               #HeadsTrayMovementStateDiagram := #"32_WIPING_POSITION_VERTICAL_WIPING";
           END_IF;
       #"32_WIPING_POSITION_VERTICAL_WIPING":
           #VerticalMotorStruct.In.RequestGoToWipingPosition := TRUE;
           IF #VerticalMotorStruct.Out.IsInWipingPosition THEN
               #VerticalMotorStruct.In.RequestGoToWipingPosition := FALSE;
               #HeadsTrayMovementStateDiagram := #"10000_MOTOR_HEADSTRAY_REQUEST_DONE";
           END_IF;

       #"40_PURGE_POSITION_VERTICAL_ORIGIN":
           #VerticalMotorStruct.In.RequestGoToOriginPosition := TRUE;
           IF #VerticalMotorStruct.Out.IsInOriginPosition THEN
               #VerticalMotorStruct.In.RequestGoToOriginPosition := FALSE;
               #HeadsTrayMovementStateDiagram := #"41_PURGE_POSITION_HORIZONTAL";
           END_IF;
       #"41_PURGE_POSITION_HORIZONTAL":
           #HorizontalMotorStruct.In.RequestGoToPurgePosition := TRUE;
           IF #HorizontalMotorStruct.Out.IsInPurgePosition THEN
               #HorizontalMotorStruct.In.RequestGoToPurgePosition := FALSE;
               #HeadsTrayMovementStateDiagram := #"42_PURGE_POSITION_VERTICAL_PURGE";
           END_IF;
       #"42_PURGE_POSITION_VERTICAL_PURGE":
           #VerticalMotorStruct.In.RequestGoToPurgePosition := TRUE;
           IF #VerticalMotorStruct.Out.IsInPurgePosition THEN
               #VerticalMotorStruct.In.RequestGoToPurgePosition := FALSE;
               #HeadsTrayMovementStateDiagram := #"10000_MOTOR_HEADSTRAY_REQUEST_DONE";
           END_IF;

       #"50_HEADS12_POSITION_VERTICAL_ORIGIN":
           #VerticalMotorStruct.In.RequestGoToOriginPosition := TRUE;
           IF #VerticalMotorStruct.Out.IsInOriginPosition THEN
               #VerticalMotorStruct.In.RequestGoToOriginPosition := FALSE;
               #HeadsTrayMovementStateDiagram := #"51_HEADS12_POSITION_HORIZONTAL";
           END_IF;
       #"51_HEADS12_POSITION_HORIZONTAL":
           #HorizontalMotorStruct.In.RequestGoToHeads12Position := TRUE;
           IF #HorizontalMotorStruct.Out.IsInHeads12Position THEN
               #HorizontalMotorStruct.In.RequestGoToHeads12Position := FALSE;
               #HeadsTrayMovementStateDiagram := #"10000_MOTOR_HEADSTRAY_REQUEST_DONE";
           END_IF;

       #"60_HEADS34_POSITION_VERTICAL_ORIGIN":
           #VerticalMotorStruct.In.RequestGoToOriginPosition := TRUE;
           IF #VerticalMotorStruct.Out.IsInOriginPosition THEN
               #VerticalMotorStruct.In.RequestGoToOriginPosition := FALSE;
               #HeadsTrayMovementStateDiagram := #"61_HEADS34_POSITION_HORIZONTAL";
           END_IF;
       #"61_HEADS34_POSITION_HORIZONTAL":
           #HorizontalMotorStruct.In.RequestGoToHeads34Position := TRUE;
           IF #HorizontalMotorStruct.Out.IsInHeads34Position THEN
               #HorizontalMotorStruct.In.RequestGoToHeads34Position := FALSE;
               #HeadsTrayMovementStateDiagram := #"10000_MOTOR_HEADSTRAY_REQUEST_DONE";
           END_IF;

       #"70_HEADS56_POSITION_VERTICAL_ORIGIN":
           #VerticalMotorStruct.In.RequestGoToOriginPosition := TRUE;
           IF #VerticalMotorStruct.Out.IsInOriginPosition THEN
               #VerticalMotorStruct.In.RequestGoToOriginPosition := FALSE;
               #HeadsTrayMovementStateDiagram := #"71_HEADS56_POSITION_HORIZONTAL";
           END_IF;
       #"71_HEADS56_POSITION_HORIZONTAL":
           #HorizontalMotorStruct.In.RequestGoToHeads56Position := TRUE;
           IF #HorizontalMotorStruct.Out.IsInHeads34Position THEN
               #HorizontalMotorStruct.In.RequestGoToHeads56Position := FALSE;
               #HeadsTrayMovementStateDiagram := #"10000_MOTOR_HEADSTRAY_REQUEST_DONE";
           END_IF;

       #"80_HIGH_POSITION_VERTICAL_ORIGIN":
           #VerticalMotorStruct.In.RequestGoToOriginPosition := TRUE;
           IF #VerticalMotorStruct.Out.IsInOriginPosition THEN
               #VerticalMotorStruct.In.RequestGoToOriginPosition := FALSE;
               #HeadsTrayMovementStateDiagram := #"81_HIGH_POSITION_HORIZONTAL_PRINTING";
           END_IF;
       #"81_HIGH_POSITION_HORIZONTAL_PRINTING":
           #HorizontalMotorStruct.In.RequestGoToPrintingPosition := TRUE;
           IF #HorizontalMotorStruct.Out.IsInPrintingPosition THEN
               #HorizontalMotorStruct.In.RequestGoToPrintingPosition := FALSE;
               #HeadsTrayMovementStateDiagram := #"10000_MOTOR_HEADSTRAY_REQUEST_DONE";
           END_IF;

       #"90_PRINT_POSITION_VERTICAL_ORIGIN":
           #VerticalMotorStruct.In.RequestGoToOriginPosition := TRUE;
           IF #VerticalMotorStruct.Out.IsInOriginPosition THEN
               #VerticalMotorStruct.In.RequestGoToOriginPosition := FALSE;
               #HeadsTrayMovementStateDiagram := #"91_PRINT_POSITION_HORIZONTAL_PRINTING";
           END_IF;
       #"91_PRINT_POSITION_HORIZONTAL_PRINTING":
           #HorizontalMotorStruct.In.RequestGoToPrintingPosition := TRUE;
           IF #HorizontalMotorStruct.Out.IsInPrintingPosition THEN
               #HorizontalMotorStruct.In.RequestGoToPrintingPosition := FALSE;
               #HeadsTrayMovementStateDiagram := #"92_PRINT_POSITION_VERTICAL_PRINTING";
           END_IF;
       #"92_PRINT_POSITION_VERTICAL_PRINTING":
           #VerticalMotorStruct.In.RequestGoToPrintingPosition := TRUE;
           IF #VerticalMotorStruct.Out.IsInPrintingPosition THEN
               #VerticalMotorStruct.In.RequestGoToPrintingPosition := FALSE;
               #HeadsTrayMovementStateDiagram := #"10000_MOTOR_HEADSTRAY_REQUEST_DONE";
           END_IF;

       #"100_VERTICAL_ORIGIN":
           #VerticalMotorStruct.In.RequestGoToOriginPosition := TRUE;
           IF #VerticalMotorStruct.Out.IsInOriginPosition THEN
               #VerticalMotorStruct.In.RequestGoToOriginPosition := FALSE;
               #HeadsTrayMovementStateDiagram := #"10000_MOTOR_HEADSTRAY_REQUEST_DONE";
           END_IF;

       #"110_VERTICAL_CLEANING":
           #VerticalMotorStruct.In.RequestGoToCleaningPosition := TRUE;
           IF #VerticalMotorStruct.Out.IsInCleaningPosition THEN
               #VerticalMotorStruct.In.RequestGoToCleaningPosition := FALSE;
               #HeadsTrayMovementStateDiagram := #"10000_MOTOR_HEADSTRAY_REQUEST_DONE";
           END_IF;
       #"10000_MOTOR_HEADSTRAY_REQUEST_DONE":
           #HorizontalMotorStruct.In.RequestHoming := FALSE;
           #HorizontalMotorStruct.In.RequestGoToOriginPosition := FALSE;
           #HorizontalMotorStruct.In.RequestGoToWipingPosition := FALSE;
           #HorizontalMotorStruct.In.RequestGoToPurgePosition := FALSE;
           #HorizontalMotorStruct.In.RequestGoToHeads12Position := FALSE;
           #HorizontalMotorStruct.In.RequestGoToHeads34Position := FALSE;
           #HorizontalMotorStruct.In.RequestGoToHeads56Position := FALSE;
           #HorizontalMotorStruct.In.RequestGoToPrintingPosition := FALSE;
           #VerticalMotorStruct.In.RequestHoming := FALSE;
           #VerticalMotorStruct.In.RequestGoToOriginPosition := FALSE;
           #VerticalMotorStruct.In.RequestGoToCleaningPosition := FALSE;
           #VerticalMotorStruct.In.RequestGoToWipingPosition := FALSE;
           #VerticalMotorStruct.In.RequestGoToPurgePosition := FALSE;
           #VerticalMotorStruct.In.RequestGoToPrintingPosition := FALSE;
           #HeadsTrayMovementStateDiagram := #"0_WAIT_FOR_MOTOR_HEADSTRAY_REQUESTS";
   END_CASE;
END_REGION

REGION Network 8 (SCL): Printing HeadsTray State Management
   //Homing
   #HeadsTray_HomingDone := #VerticalMotorStruct.Out.HomingDone AND #HorizontalMotorStruct.Out.HomingDone;

   //Actual Position
   #VerticalMotor_ActualPosition_mm := #VerticalMotorStruct.Out.ActualPosition;
   #HorizontalMotor_ActualPosition_mm := #HorizontalMotorStruct.Out.ActualPosition;

   //Vertical Motor Position
   #VerticalMotor_IsInOriginPosition := #VerticalMotorStruct.Out.IsInOriginPosition;
   #VerticalMotor_IsInWipingPosition := #VerticalMotorStruct.Out.IsInWipingPosition;
   #VerticalMotor_IsInPurgePosition := #VerticalMotorStruct.Out.IsInPurgePosition;
   #VerticalMotor_IsInCleaningPosition := #VerticalMotorStruct.Out.IsInCleaningPosition;
   #VerticalMotor_IsInPrintingPosition := #VerticalMotorStruct.Out.IsInPrintingPosition;

   //Horizontal Motor Position
   #HorizontalMotor_IsInOriginPosition := #HorizontalMotorStruct.Out.IsInOriginPosition;
   #HorizontalMotor_IsInWipingPosition := #HorizontalMotorStruct.Out.IsInWipingPosition;
   #HorizontalMotor_IsInPurgePosition := #HorizontalMotorStruct.Out.IsInPurgePosition;
   #HorizontalMotor_IsInHeads12Position := #HorizontalMotorStruct.Out.IsInHeads12Position;
   #HorizontalMotor_IsInHeads34Position := #HorizontalMotorStruct.Out.IsInHeads34Position;
   #HorizontalMotor_IsInHeads56Position := #HorizontalMotorStruct.Out.IsInHeads56Position;
   #HorizontalMotor_IsInPrintingPosition := #HorizontalMotorStruct.Out.IsInPrintingPosition;

   //HeadsTray Position
   #HeadsTray_IsInOriginPosition := #HorizontalMotor_IsInOriginPosition AND #VerticalMotor_IsInOriginPosition;
   #HeadsTray_IsInWipingPosition := #HorizontalMotor_IsInOriginPosition AND #VerticalMotor_IsInWipingPosition;
   #HeadsTray_IsInHeads12CleaningPosition := #HorizontalMotor_IsInHeads12Position AND #VerticalMotor_IsInCleaningPosition;
   #HeadsTray_IsInHeads34CleaningPosition := #HorizontalMotor_IsInHeads34Position AND #VerticalMotor_IsInCleaningPosition;
   #HeadsTray_IsInHeads56CleaningPosition := #HorizontalMotor_IsInHeads56Position AND #VerticalMotor_IsInCleaningPosition;
   #HeadsTray_IsInPurgePosition := #HorizontalMotor_IsInOriginPosition AND #VerticalMotor_IsInPurgePosition;
   #HeadsTray_IsInHighPosition := #HorizontalMotor_IsInPrintingPosition AND #VerticalMotor_IsInOriginPosition;
   #HeadsTray_IsInPrintingPosition := #HorizontalMotor_IsInPrintingPosition AND #VerticalMotor_IsInPrintingPosition;

   //Error
   #VerticalMotor_InError := #VerticalMotorStruct.Out.InError;
   #VerticalMotor_ErrorCode := #VerticalMotorStruct.Out.ErrorCode;
   #HorizontalMotor_InError := #HorizontalMotorStruct.Out.InError;
   #HorizontalMotor_ErrorCode := #HorizontalMotorStruct.Out.ErrorCode;
END_REGION
END_FUNCTION_BLOCK
